FUNCTION_BLOCK GoToAuto IMPLEMENTS I_Transitive
VAR
    _currentState : POINTER TO I_SD_ValveState;
    _nextState : REFERENCE TO AutoState;
END_VAR

METHOD FB_init : BOOL
VAR_INPUT
	bInitRetains : BOOL; // if TRUE, the retain variables are initialized (warm start / cold start)
	bInCopyCode : BOOL;  // if TRUE, the instance afterwards gets moved into the copy code (online change)
    currentState : POINTER TO I_SD_ValveState;
    nextState : REFERENCE TO AutoState;
END_VAR
_currentState := currentState;
_nextState REF= nextState;
END_METHOD

METHOD Transit
_currentState^ := _nextState;
END_METHOD

END_FUNCTION_BLOCK

(* stored: Version 1.1.0.1, ProductVersion 3.1.4024.12
   POU GoToAuto: Id {2fd6b091-f1dd-4786-b628-fdd42456d316}, SpecialFunc None
   Method FB_init: Id {33f411ab-54fd-4e32-b517-194ad46909a8}
   Method Transit: Id {e1e220d0-c8c0-4051-acfa-07426ddde60e} *)
